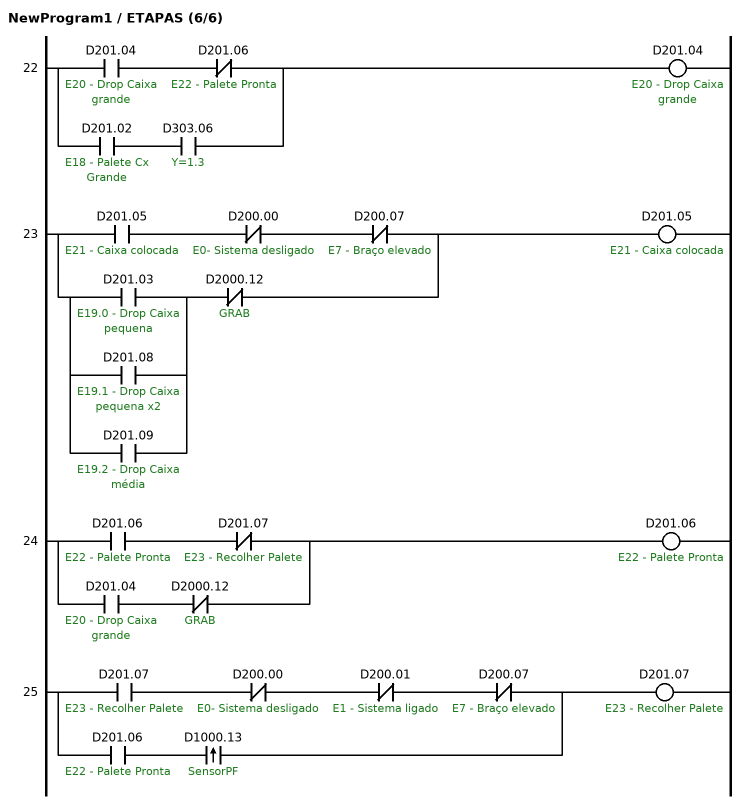
; [picture p24: NewProgram1 / ETAPAS, rungs 22-25]
; rung 22
LD D201.04  ; E20 - Drop Caixa grande
ANDNOT D201.06  ; E22 - Palete Pronta
LD D201.02  ; E18 - Palete Cx Grande
AND D303.06  ; Y=1.3
ORLD
OUT D201.04  ; E20 - Drop Caixa grande
; rung 23
LD D201.05  ; E21 - Caixa colocada
ANDNOT D200.00  ; E0- Sistema desligado
ANDNOT D200.07  ; E7 - Braço elevado
LD D201.03  ; E19.0 - Drop Caixa pequena
OR D201.08  ; E19.1 - Drop Caixa pequena x2
OR D201.09  ; E19.2 - Drop Caixa média
ANDNOT D2000.12  ; GRAB
ORLD
OUT D201.05  ; E21 - Caixa colocada
; rung 24
LD D201.06  ; E22 - Palete Pronta
ANDNOT D201.07  ; E23 - Recolher Palete
LD D201.04  ; E20 - Drop Caixa grande
ANDNOT D2000.12  ; GRAB
ORLD
OUT D201.06  ; E22 - Palete Pronta
; rung 25
LD D201.07  ; E23 - Recolher Palete
ANDNOT D200.00  ; E0- Sistema desligado
ANDNOT D200.01  ; E1 - Sistema ligado
ANDNOT D200.07  ; E7 - Braço elevado
LD D201.06  ; E22 - Palete Pronta
@AND D1000.13  ; SensorPF
ORLD
OUT D201.07  ; E23 - Recolher Palete

### Section END
; rung 0
END(001)